Staubli VAL3: refreshDynamic.pgx

program refreshDynamic()
begin
  // DO NOT CHANGE
  nRefresh=clock()
  //
  // ADD HERE
  //
  use:bUseRefresh=false
end
